PROGRAM MAIN
VAR
	Hello :BOOL;
	ScopeTrigger: BOOL;
	

	Baseline: INT;
END_VAR





fast();

Laser();

YaxisBar();

Velocimeter();

ReelCommand();

VariableTesting();

Baseline := -20;


IF bSet OR bSetBTN THEN
	veloreset	:= TRUE;
	
	ELSE 
	veloreset	:= FALSE;	
	
	
END_IF

END_PROGRAM

(* stored: Version 1.1.0.1, ProductVersion 3.1.4024.12
   POU MAIN: Id {42181531-c32c-4115-8b0f-9c27bdf5888c}, SpecialFunc None *)
